GLOBALCONSTANTS DefaultPool_PWM_Numeric (* Numeric object pool constants (ID, Scale, Offset, Decimals) *)
  PACKAGE Uebungen::const::UT::PWM;
  VAR_GLOBAL CONSTANT
    InputNumber_PWM_DUTY : logiBUS::utils::conversion::phys::NumericObjectPool_S := (u16ObjId := 9000, r32Scale := 0.0122085215, i32Offset := 0, u8Decimals := 3);
    NumberVariable_PWM_Value : logiBUS::utils::conversion::phys::NumericObjectPool_S := (u16ObjId := 9000, r32Scale := 0.0122085215, i32Offset := 0, u8Decimals := 3);
    InputNumber_PWM_Value : logiBUS::utils::conversion::phys::NumericObjectPool_S := (u16ObjId := 9001, r32Scale := 1.0, i32Offset := 0, u8Decimals := 0);
    InputNumber_PWM_DUTY_OUT : logiBUS::utils::conversion::phys::NumericObjectPool_S := (u16ObjId := 9002, r32Scale := 0.0122085215, i32Offset := 0, u8Decimals := 3);
    InputNumber_THRESHOLD : logiBUS::utils::conversion::phys::NumericObjectPool_S := (u16ObjId := 9003, r32Scale := 0.0122085215, i32Offset := 0, u8Decimals := 3);
    InputNumber_HYSTERESIS : logiBUS::utils::conversion::phys::NumericObjectPool_S := (u16ObjId := 9004, r32Scale := 0.0122085215, i32Offset := 0, u8Decimals := 3);
    OutputNumber_100 : logiBUS::utils::conversion::phys::NumericObjectPool_S := (u16ObjId := 12000, r32Scale := 1.0, i32Offset := 0, u8Decimals := 0);
    OutputNumber_8129 : logiBUS::utils::conversion::phys::NumericObjectPool_S := (u16ObjId := 12001, r32Scale := 1.0, i32Offset := 0, u8Decimals := 0);
    OutputNumber_050 : logiBUS::utils::conversion::phys::NumericObjectPool_S := (u16ObjId := 12002, r32Scale := 1.0, i32Offset := 0, u8Decimals := 0);
    OutputNumber_075 : logiBUS::utils::conversion::phys::NumericObjectPool_S := (u16ObjId := 12003, r32Scale := 1.0, i32Offset := 0, u8Decimals := 0);
    OutputNumber_000 : logiBUS::utils::conversion::phys::NumericObjectPool_S := (u16ObjId := 12004, r32Scale := 1.0, i32Offset := 0, u8Decimals := 0);
    OutputNumber_025 : logiBUS::utils::conversion::phys::NumericObjectPool_S := (u16ObjId := 12005, r32Scale := 1.0, i32Offset := 0, u8Decimals := 0);
  END_VAR
END_GLOBALCONSTANTS
